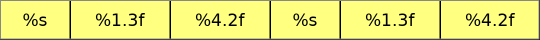
VISUALIZATION VISU_CONFIG_LIGNE_GAZ_SEUIL  // 540x40
VAR_IN_OUT
	m_Input_MASSFLOW:		BLOCK_MFC_BROOKS_NoCoE;
END_VAR
    Rectangle (70,0 100x40), "%1.3f", text variable: m_Input_MASSFLOW.CONF_Nom_Coef, input disabled if: NOT Global_Variables.PRG_USER.ACTU_USER.CONF_MACHINE
        OnMouseDown: write the text variable via InputWithLimits
    Rectangle (170,0 100x40), "%4.2f", text variable: m_Input_MASSFLOW.CONF_Nom_max_flow, input disabled if: NOT Global_Variables.PRG_USER.ACTU_USER.CONF_MACHINE
        OnMouseDown: write the text variable via InputWithLimits
    Rectangle (340,0 100x40), "%1.3f", text variable: m_Input_MASSFLOW.CONF_Util_Coef, input disabled if: NOT Global_Variables.PRG_USER.ACTU_USER.CONF_MACHINE
        OnMouseDown: write the text variable via InputWithLimits
    Rectangle (440,0 100x40), "%4.2f", text variable: m_Input_MASSFLOW.CONF_Util_Max_Flow, input disabled if: NOT Global_Variables.PRG_USER.ACTU_USER.CONF_MACHINE
    Rectangle (0,0 70x40), "%s", text variable: m_Input_MASSFLOW.CONF_Nom_Name, input disabled if: NOT Global_Variables.PRG_USER.ACTU_USER.CONF_MACHINE
        OnMouseDown: write the text variable via InputWithLimits
    Rectangle (270,0 70x40), "%s", text variable: m_Input_MASSFLOW.CONF_Util_Name, input disabled if: NOT Global_Variables.PRG_USER.ACTU_USER.CONF_MACHINE
        OnMouseDown: write the text variable via InputWithLimits
END_VISUALIZATION

(* stored: Version 1.1.0.1, ProductVersion 3.1.4024.10
   Visu VISU_CONFIG_LIGNE_GAZ_SEUIL: Id {31f2ae93-c406-4758-bcd9-ecc7e4ea7028} *)
